{attribute 'pack_mode' := '1'}
TYPE
BuR_MoverAxis_EtherCAT_st :
STRUCT
    diCurrentPos_um   : DINT; (* current position, expressed as um *)
    iCurrentVelo_mmps : INT;  (* current velocity in mm per second *)
    bStatus           : UINT; (* status flag                       *)
    bShelfLentgh_mm   : INT;  (* shelf length in mm                *)
END_STRUCT
END_TYPE

(* stored: Version 1.1.0.1, ProductVersion 3.1.4024.6
   DUT BuR_MoverAxis_EtherCAT_st: Id {64ae641a-6eb5-4916-a008-7abaf4789670} *)
